# EPICS substitutions: enginxJawsApp/Db/enginxjawset.substitutions
file enginxjawset.template {
  pattern
    {DIR,           dir_name,		P,       JAWS,			MTR,  		HIGH_GAP_LIMIT, LOW_GAP_LIMIT, 		MTR_TO_GAP_A, 	MTR_TO_GAP_B, 	MTR_TO_GAP_C,			MTR_FRM_GAP_A, 	MTR_FRM_GAP_B, 	MTR_FRM_GAP_C}
    {"V", 		"Vertical",		"\$(P)", "\$(JAWS)",	"\$(NS_MTR)", 	"25", 			"0.5", 				-0.0358, 		2.0167,			-2.0091, 				0.0138,			0.4146,			1.1885}
    {"H", 		"Horizontal",	"\$(P)", "\$(JAWS)",	"\$(EW_MTR)", 	"10", 			"0.5",				0.0434,			-0.4519,		0.8232,  				-0.0776,		1.9001,			8.9105}
}
